// TwinCAT 3 PLC project Plc
// ProgramVersion: 3.1.4023.0
// libraries:
//   Tc2_Standard, * (Beckhoff Automation GmbH)
//   Tc2_System, * (Beckhoff Automation GmbH)
//   Tc3_EventLogger, * (Beckhoff Automation GmbH)
//   Tc3_Module, * (Beckhoff Automation GmbH)
// project tree:
//   DUTs/ ST_MyType.TcDUT
//   / PlcTask.TcTTO
//   POUs/ AlarmExtension.TcPOU, Alarming.TcPOU, AlarmingEx.TcPOU, MAIN.TcPOU
// real-time tasks:
//   TASK PlcTask: cycle T#10ms, priority 20, ADS port 350

CONFIGURATION Plc
    RESOURCE PLC ON TwinCAT3
        TASK PlcTask(INTERVAL := T#10ms, PRIORITY := 20);
        PROGRAM MAIN WITH PlcTask : MAIN;
    END_RESOURCE
END_CONFIGURATION

// ---- DUTs/ST_MyType.TcDUT
TYPE ST_MyType :
STRUCT
	bValue	: BOOL;
	iValue	: INT;
	sValue	: STRING;
END_STRUCT
END_TYPE

// ---- POUs/MAIN.TcPOU
PROGRAM MAIN
VAR
	iCounter : INT;
	bToggle		: BOOL;
	bReset		: BOOL;
	sText		: STRING;
	
	stMyType		: ST_MyType;
	
END_VAR


IF bToggle THEN
	sText := 'stop';
	iCounter := (iCounter + 1) MOD 1000;
	IF iCounter = 0 THEN
		bToggle := FALSE;
	END_IF
ELSE
	sText := 'start';
	IF bReset THEN
		bReset := FALSE;
		iCounter := 0;
	END_IF	
END_IF

Alarming();
AlarmingEx();
AlarmExtension();

END_PROGRAM

// ---- POUs/Alarming.TcPOU
PROGRAM Alarming
VAR
	bInit 		: BOOL := TRUE;
	bSendMsg	: BOOL;
	fbMsg		: FB_TcMessage;
END_VAR

IF bInit THEN
	bInit := FALSE;
	fbMsg.CreateEx(TC_Events.MyEventClass.MyMessage, 0);
END_IF

IF bSendMsg THEN
	bSendMsg := FALSE;
	fbMsg.Send(0);
END_IF

END_PROGRAM

// ---- POUs/AlarmingEx.TcPOU
PROGRAM AlarmingEx
VAR
	bInit			: BOOL := TRUE;
	bRaise			: BOOL;
	bClear			: BOOL;
	
	fbAlm			: FB_TcAlarm;
	fbSourceInfo	: FB_TcSourceInfo;
END_VAR

IF bInit THEN
	bInit := FALSE;
	
	fbSourceInfo.Clear();
	fbSourceInfo.sName := '%l%L_MyName%/l%';
	
	//fbAlm.CreateEx(TC_Events.MyEventClass.MyAlarm, TRUE, 0);
	fbAlm.CreateEx(TC_Events.MyEventClass.MyAlarm, TRUE, fbSourceInfo);
	
	fbAlm.ipArguments.Clear();
	fbAlm.ipArguments.AddString('BMK');
END_IF

IF bRaise THEN
	bRaise := FALSE;
	fbAlm.Raise(0);
END_IF

IF bClear AND (fbAlm.eConfirmationState = TcEventConfirmationState.Confirmed) THEN
	bClear := FALSE;
	fbAlm.Clear(0, FALSE);
END_IF

END_PROGRAM

// ---- POUs/AlarmExtension.TcPOU
PROGRAM AlarmExtension
VAR
	bAlarm		: BOOL;
	iAlarm		: INT;
END_VAR

END_PROGRAM
